{attribute 'linkalways'} 
{attribute 'no_explicit_call' := 'This FB is a CLASS and must be accessed using methods or properties'}
{attribute 'enable_dynamic_creation'}
FUNCTION_BLOCK Node_ContainerType_Vector_TcVnVector3_USINT EXTENDS Node
VAR
    out : _GUID;
END_VAR

METHOD PUBLIC  Clone : I_Node
VAR
	pNode : POINTER TO Node_ContainerType_Vector_TcVnVector3_USINT;
END_VAR
pNode := __NEW(Node_ContainerType_Vector_TcVnVector3_USINT);
Clone := pNode^;
END_METHOD

METHOD FB_init : BOOL
VAR_INPUT
	bInitRetains : BOOL; // if TRUE, the retain variables are initialized (warm start / cold start)
	bInCopyCode : BOOL;  // if TRUE, the instance afterwards gets moved into the copy code (online change)
END_VAR
AddOutput('out', out);
END_METHOD

METHOD PROTECTED OnExecute
out.Value := ContainerType_Vector_TcVnVector3_USINT;
END_METHOD

END_FUNCTION_BLOCK

(* stored: Version 1.1.0.1, ProductVersion 3.1.4026.17
   POU Node_ContainerType_Vector_TcVnVector3_USINT: Id {eeb35fdb-7162-06b1-12aa-1cad53bc49a0}, SpecialFunc None
   Folder Constructor: Id {c8db8470-2d1e-0a54-283b-6c1d0900e9ef}
   Method Clone: Id {a676bc0e-21dc-0198-195c-13f7bf8af1aa}
   Method FB_init: Id {b31f4745-d39f-0fb3-11a2-66e132fff464}
   Method OnExecute: Id {57ce4b68-08eb-0cf1-1301-9fdea0eb01f6} *)
